FUNCTION_BLOCK overcurrentV2_IO_1 (* Composite Function Block Type *)
  (* Standard: 61499-2 *)
  (* Version 0.0, 23/05/2016, Chen-Wei, nxtControl GmbH, template *)
  PACKAGE Main;
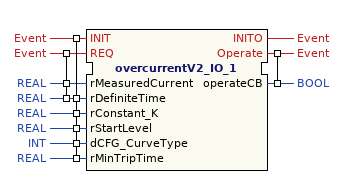
  EVENT_INPUT
    INIT WITH rDefiniteTime, rConstant_K, rStartLevel, dCFG_CurveType, rMinTripTime; (* Initialization Request *)
    REQ WITH rMeasuredCurrent, rDefiniteTime; (* Normal Execution Request *)
  END_EVENT
  EVENT_OUTPUT
    INITO; (* Initialization Confirm *)
    Operate WITH operateCB; (* Delayed Event *)
  END_EVENT
  VAR_INPUT
    rMeasuredCurrent : REAL; (* Input event qualifier *)
    rDefiniteTime : REAL;
    rConstant_K : REAL;
    rStartLevel : REAL;
    dCFG_CurveType : INT;
    rMinTripTime : REAL;
  END_VAR
  VAR_OUTPUT
    operateCB : BOOL; (* Output event qualifier *)
  END_VAR
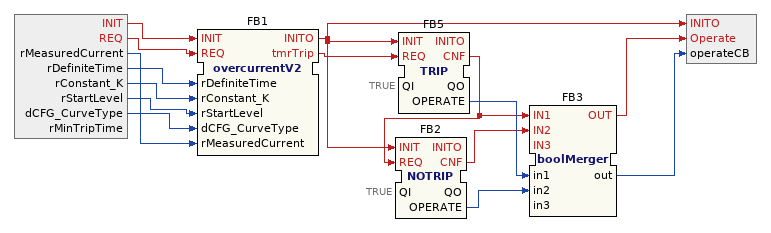
  FBS
    FB5 : TRIP(QI := TRUE);
    FB1 : overcurrentV2;
    FB2 : NOTRIP(QI := TRUE);
    FB3 : boolMerger;
  END_FBS
  EVENT_CONNECTIONS
    INIT TO FB1.INIT;
    REQ TO FB1.REQ;
    FB1.INITO TO INITO;
    FB1.tmrTrip TO FB5.REQ;
    FB1.INITO TO FB5.INIT;
    FB5.CNF TO FB3.IN1;
    FB2.CNF TO FB3.IN2;
    FB3.OUT TO Operate;
    FB1.INITO TO FB2.INIT;
    FB5.CNF TO FB2.REQ;
  END_CONNECTIONS
  DATA_CONNECTIONS
    rDefiniteTime TO FB1.rDefiniteTime;
    rConstant_K TO FB1.rConstant_K;
    rStartLevel TO FB1.rStartLevel;
    dCFG_CurveType TO FB1.dCFG_CurveType;
    rMeasuredCurrent TO FB1.rMeasuredCurrent;
    FB5.OPERATE TO FB3.in1;
    FB2.OPERATE TO FB3.in2;
    FB3.out TO operateCB;
  END_CONNECTIONS
END_FUNCTION_BLOCK
